KUKA KRL data list: git_clean_demo.dat

&ACCESS RVP
&REL 48
&COMMENT WorkVisual Header DAT
&PARAM EDITMASK = *
DEFDAT git_clean_demo
  DECL INT nVersion = 48
ENDDAT
